Fanuc TP program (LS listing): MOVETOMAINT3.LS

/PROG  MOVETOMAINT3
/ATTR
OWNER		= MNEDITOR;
COMMENT		= "";
PROG_SIZE	= 421;
CREATE		= DATE 18-04-17  TIME 08:11:34;
MODIFIED	= DATE 18-04-19  TIME 06:45:26;
FILE_NAME	= MOVETOMA;
VERSION		= 0;
LINE_COUNT	= 15;
MEMORY_SIZE	= 865;
PROTECT		= READ;
TCD:  STACK_SIZE	= 0,
      TASK_PRIORITY	= 50,
      TIME_SLICE	= 0,
      BUSY_LAMP_OFF	= 0,
      ABORT_REQUEST	= 0,
      PAUSE_REQUEST	= 0;
DEFAULT_GROUP	= 1,*,*,*,*;
CONTROL_CODE	= 00000000 00000000;
/APPL

AUTO_SINGULARITY_HEADER;
  ENABLE_SINGULARITY_AVOIDANCE   : FALSE;
/MN
   1:  !move to maint ;
   2:   ;
   3:  UFRAME_NUM=0 ;
   4:  UTOOL_NUM=3 ;
   5:   ;
   6:  !if at another maint pos ;
   7:  IF DO[100:OFF:At Maint 1]=ON OR DO[101:OFF:At Maint 2]=ON,JMP LBL[10] ;
   8:   ;
   9:   ;
  10:J PR[35:Pallet 4&5SafePt] 25% CNT100    ;
  11:   ;
  12:  LBL[10] ;
  13:J PR[57:maint 3] 25% FINE    ;
  14:   ;
  15:   ;
/POS
/END
